PROGRAM PRG_Puls
VAR
	    //=== Master Pulses ===//
	fbScalingFlash  :FB_Pulse;
	fbScalingFlash4 :FB_Pulse;
	fbScalingFlash5 :FB_Pulse;
	fbFlash100Hz    :FB_Pulse;
	fbFlash10Hz		:FB_Pulse;
	fbFlash10HzB    :FB_Pulse;
	fbFlash4Hz		:FB_Pulse;
	fbFlash2Hz		:FB_Pulse;
	fbFlash1Hz		:FB_Pulse;
    fbFlash5Sec     :FB_Pulse;			

END_VAR

    //=== Master Pulses ===//
(**************************************************************************************************)
fbScalingFlash(
	bEnable	:=	TRUE,
	tPulseOn	:=	T#2MS,
	tPulseOff	:=	T#2MS,
	bFlash		=>	stPuls.bFlashScale
);

fbScalingFlash4(
     bEnable	:=	TRUE,
	tPulseOn	:=	T#4MS,
	tPulseOff	:=	T#4MS,
	bFlash		=>	stPuls.bFlashScale4
);
fbScalingFlash5(
     bEnable	:=	TRUE,
	tPulseOn	:=	T#5MS,
	tPulseOff	:=	T#5MS,
	bFlash		=>	stPuls.bFlashScale5
);



fbFlash100Hz(
	bEnable	:=	TRUE,
	tPulseOn	:=	T#10MS,
	tPulseOff	:=	T#10MS,
	bFlash		=>	stPuls.bFlash100Hz
);


fbFlash10HzB ( 
    bEnable	    :=	TRUE,
	tPulseOn	:=	T#20MS,//  T#50MS,
	tPulseOff	:=	T#20MS,//  T#50MS,
	bFlash		=>	stPuls.bFlash10BHz
);


fbFlash10Hz(
	bEnable	:=	TRUE,
	tPulseOn	:=	T#100MS,
	tPulseOff	:=	T#100MS,
	bFlash		=>	stPuls.bFlash10Hz
);


fbFlash4Hz(
	bEnable	:=	TRUE,
	tPulseOn	:=	T#250MS,
	tPulseOff	:=	T#250MS,
	bFlash		=>	stPuls.bFlash4Hz
);

fbFlash2Hz(
	bEnable	:=	TRUE,
	tPulseOn	:=	T#500MS,
	tPulseOff	:=	T#500MS,
	bFlash		=>	stPuls.bFlash2Hz
);

fbFlash1Hz(
	bEnable	:=	TRUE,
	tPulseOn	:=	T#1000MS,
	tPulseOff	:=	T#1000MS,
	bFlash		=>	stPuls.bFlash1Hz
);

fbFlash5Sec(
	bEnable	:=	TRUE,
	tPulseOn	:=	T#5S,
	tPulseOff	:=	T#5S,
	bFlash		=>	stPuls.bFlash5sec
);

END_PROGRAM

(* stored: Version 1.1.0.1, ProductVersion 3.1.4024.13
   POU PRG_Puls: Id {41f93764-460c-4865-ba92-1d1cdc722a5e}, SpecialFunc None *)
